PROGRAM Run
VAR	
	buffer					: ARRAY[1..4096] OF BYTE;
	path					: MC_PATH_DATA_REF(ADR(buffer), SIZEOF(buffer));
	
	aTargetPos				: ARRAY[1..cAxesCount] OF MC_LREAL;
	aTransitionParam		: ARRAY[1..2] OF MC_LREAL;
	
	fVelFactor				: LREAL := 1.0;
	
	fbPower					: FB_EnableAxes;
	fbAddAllAxes			: FB_AddAllAxes;
	fbGroupEnable			: MC_GroupEnable;
	fbMoveLinPrep			: MC_MoveLinearAbsolutePreparation;
	fbMovePath				: MC_MovePath;
	fbStop					: MC_GroupStop;
	fbUngroupAxes			: MC_UngroupAllAxes;
	fbGroupReset			: MC_GroupReset;
	fbGroupReadStatus		: MC_GroupReadStatus;
	fbGroupSetOvr			: MC_GroupSetOverride;
	
	nState					: INT := -5;
	nNextState				: INT;
	bMovePrepError			: BOOL;
	bPickCycle				: BOOL;
	bExecutePath			: BOOL := TRUE;
	
	bUserIncrementStep		: BOOL; // user can go to next step
	bUserInfiniteMovement 	: BOOL := TRUE; // user can decide if only one movement is executed or infinite movement.
	bUserStop				: BOOL; // user triggered stop
	bUserForceUngroup		: BOOL; // user triggered ungroup axes
	bUserForceReset			: BOOL; // user triggered reset
	
	
	
	
	bUserEnableAxes:	BOOL:= TRUE;
	bUserConfigGroup:	BOOL	:= FALSE;
	bUserCartesianMode:	BOOL	:= TRUE;
	bUserResetKinGroup:	BOOL	:= FALSE;		
	
	in_stKinToPlc	AT %I*:	NcToPlc_NciChannel_Ref;
	in_stItpToPlc	AT %I*:	NcToPlc_NciChannel_Ref;
	out_stPlcToKin	AT %Q*:	PLCTONC_NCICHANNEL_REF;
	out_stPlcToItp	AT %Q*:	PLCTONC_NCICHANNEL_REF;
	
	//:	FB_EnableAxes;
	bAllAxesReady:	BOOL;
	
	stAxesConfig:	ST_KinAxes;
	fbConfigKinGroup:	FB_KinConfigGroup;
	fbResetKinGroup:	FB_KinResetGroup;
	
	//MODDED CODE VARIABLES
	frameHome : StructFrame := (rXpos := 0, rXpos := 0, rZpos := 147.0, sAlias := 'Home');
	iFrameSequence : INT := 0;
	bRunSequence: BOOL;
	
	
	//////////////
	//Reset
	bResetNC: BOOL;
	bKinFactoryReset: BOOL;
	bResetKinGrp: BOOL;
	nReset: INT;
	nKinReset: INT;
	nGroupReset: INT;
	bKinResetDone: BOOL;
	bGroupResetDone: BOOL;
	fbNCReset	: FB_NCReset;
	bInitMove : BOOL := TRUE;
	iInterpolation : INT := 1;
	bRepeat : BOOL := FALSE;
	
	timerDisable: TON;
	bMagnet: BOOL;
	bXbox : BOOL;
	controller: xbox;
	frameNow: StructFrame;
	frameTarget: StructFrame;
	bAnyBtn : BOOL;
END_VAR

VAR_INPUT
	arrangedFrames : ARRAY [0..20] OF StructFrame;
	nManual: INT;
END_VAR

//==========================================
// PnpSimpleSample V1.3
//==========================================

//==========================================
//	Set variable bUserIncrementStep:= TRUE to go to the next step
//	Variable bUserInfiniteMovement defines if only one movement or infinite
//	movement is executed.
//==========================================



fbGroupReadStatus(
	AxesGroup:= stGroupRef , 
	Enable:= TRUE , 
	Valid=> , 
	Busy=> , 
	GroupMoving=> , 
	GroupHoming=> , 
	GroupErrorStop=> , 
	GroupNotReady=> , 
	GroupStandby=> , 
	GroupStopping=> , 
	GroupDisabled=> , 
	Error=> , 
	ErrorId=> );
IF fbGroupReadStatus.Error THEN
	nState := 9998;
ELSIF NOT fbGroupReadStatus.Valid THEN
	nState := 9999;	
END_IF

fbGroupSetOvr(
	AxesGroup:= stGroupRef, 
	Enable:= TRUE, 
	VelFactor:= fVelFactor , 
	Enabled=> , 
	Busy=> , 
	Error=> , 
	ErrorId=> , 
	ActualVelFactor=> );

IF fbGroupSetOvr.Error THEN
	nState := 9999;
END_IF
	
	


fbPower(
	io_X:= stAxis[1],
	io_Y:= stAxis[2],
	io_Z:= stAxis[3],
	//io_C:= stAxis[4],
	io_M1:= stACSAxis[1],
	io_M2:= stACSAxis[2],
	io_M3:= stACSAxis[3],);
	

stAxesConfig.nAxisIdsAcs[1]	:= stACSAxis[1].NcToPlc.AxisId;
stAxesConfig.nAxisIdsAcs[2]	:= stACSAxis[2].NcToPlc.AxisId;
stAxesConfig.nAxisIdsAcs[3]	:= stACSAxis[3].NcToPlc.AxisId;
stAxesConfig.nAxisIdsMcs[1]	:= stAxis[1].NcToPlc.AxisId;
stAxesConfig.nAxisIdsMcs[2]	:= stAxis[2].NcToPlc.AxisId;
stAxesConfig.nAxisIdsMcs[3]	:= stAxis[3].NcToPlc.AxisId;	
	

CASE nState OF
-5:
	IF bUserIncrementStep THEN
		nNextState := nState +1; 
		nState := 101;
		fbAddAllAxes(Execute:= FALSE);
		fbGroupEnable(AxesGroup:=stGroupRef , Execute:=FALSE);
		fbMovePath(AxesGroup:=stGroupRef ,PathData:=path ,Execute:= FALSE);
		bMovePrepError := FALSE;
	END_IF
-4:	
	fbPower.bEnableAxes := TRUE;
	
	IF fbPower.bAllAxesReady THEN
		IF bUserIncrementStep THEN
			nNextState := nState +1;
			nState := 101;
		END_IF
	ELSIF	fbPower.Error THEN
		nState := nState +1000;	
	END_IF
	
-3:
	fbConfigKinGroup(
		bExecute:=bUserConfigGroup , 
		bCartesianMode:=bUserCartesianMode , 
		stAxesList:=stAxesConfig , 
		stKinRefIn:= in_stKinToPlc, 
		bBusy=> , 
		bDone=> , 
		bError=> , 
		nErrorId=> );
	
	fbResetKinGroup(
		bExecute:=bUserResetKinGroup, 
		nItpChannelId:=0 , 
		stKinRefIn:=in_stKinToPlc, 
		stAxesList:=stAxesConfig, 
		bBusy=> , 
		bDone=> , 
		bError=> , 
		nErrorId=> );
		
	IF fbConfigKinGroup.bDone AND fbResetKinGroup.bDone THEN
		nNextState:= nState + 1;
		nState:= 101;
	ELSIF fbConfigKinGroup.bError OR fbResetKinGroup.bError THEN
		nState:= nState + 1000;
	END_IF
	
-2:
	//Add all axes to group
	fbAddAllAxes(Execute:= TRUE);
	
	IF fbAddAllAxes.Done THEN
		IF bUserIncrementStep THEN
			fbAddAllAxes(Execute:= FALSE);
			nNextState := nState +1;
			nState := 101;
		END_IF
	ELSIF fbAddAllAxes.Error THEN
		nState := nState +1000;
	END_IF
	
-1:	
	//Enable Group
	fbGroupEnable(AxesGroup:=stGroupRef , Execute:=TRUE);
	 
	IF fbGroupEnable.Done THEN
		IF bUserIncrementStep THEN
			fbGroupEnable(AxesGroup:=stGroupRef , Execute:=FALSE);
			nNextState := nState +1;
			nState := 101;
		END_IF
	ELSIF fbGroupEnable.Error THEN
		nState := nState +1000;
	END_IF
0:
	//Fill path table and start execution with fbMovePath
	IF bUserIncrementStep OR bUserInfiniteMovement THEN
		(*IF bPickCycle THEN 
			//Prepare table (MC_MoveLinearAbsolutePreparation)
			A_PreparePathPick();
		ELSE
			//Prepare table (MC_MoveLinearAbsolutePreparation)	
			A_PreparePathPlace();
		END_IF		
		bPickCycle := NOT bPickCycle;*)
		IF bRunSequence THEN
			frameNow.rXpos  := GVL.stAxis[1].NcToPlc.ActPos;
			frameNow.rYpos  := GVL.stAxis[2].NcToPlc.ActPos;
			frameNow.rZpos  := GVL.stAxis[3].NcToPlc.ActPos;
			frameTarget := frameNow;
			END_IF
			
			IF controller.bDpadUp THEN
				//frameTarget := frameNow;
				frameTarget.rYpos := frameNow.rYpos + 1;
				END_IF
			
			IF controller.bDpadDown THEN
				//frameTarget := frameNow;
				frameTarget.rYpos := frameNow.rYpos - 1;
				END_IF
			
			IF controller.bDpadLeft THEN
				//frameTarget := frameNow;
				frameTarget.rXpos := frameNow.rXpos + 1;
				END_IF
			
			IF controller.bDpadRight THEN
				//frameTarget := frameNow;
				frameTarget.rXpos := frameNow.rXpos - 1;
				END_IF
				
			IF controller.bYbtn THEN
				//frameTarget := frameNow;
				frameTarget.rZpos := frameNow.rZpos + 1;
				END_IF
				
			IF controller.bAbtn THEN
				//frameTarget := frameNow;
				frameTarget.rZpos := frameNow.rZpos - 1;
				END_IF
				
			bAnyBtn := (controller.bDpadDown OR controller.bDpadLeft OR controller.bDpadUp OR
						 controller.bDpadRight OR controller.bYbtn OR controller.bAbtn);
			
			IF bAnyBtn THEN
				MoveToPositionGeneral(currentFrame := frameNow, targetFrame := frameTarget, interpolation := 1);
				fbMovePath(AxesGroup:= stGroupRef, PathData:= path, Execute:= TRUE);

				IF bMovePrepError THEN
					nState := nState +1000;
				ELSE
					IF fbMovePath.Done THEN
						fbMovePath(AxesGroup:= stGroupRef, PathData:= path, Execute:= FALSE);
						IF bUserInfiniteMovement THEN
							nState := nState +1;
						ELSIF bUserIncrementStep THEN
							nNextState := nState + 1;
							nState := 101;
						END_IF
					END_IF
				END_IF	
			END_IF			
		END_IF

1:
	//Execute prepared movement
	fbMovePath(
		AxesGroup:= stGroupRef , 
		PathData:= path , 
		Execute:= bExecutePath
	);
	
	IF fbMovePath.Done THEN
		IF bUserIncrementStep THEN
			//ungroup axes
			nNextState := 50;
			nState := 101;
			fbMovePath(AxesGroup:= stGroupRef, PathData:= path, Execute:= FALSE);
		ELSIF bUserInfiniteMovement THEN
			nState := nState -1;
			fbMovePath(AxesGroup:= stGroupRef, PathData:= path, Execute:= FALSE);
		END_IF
	ELSIF fbMovePath.Error THEN
		nState := nState + 1000;	
	END_IF
20:
	fbStop(AxesGroup:=stGroupRef, Execute:= FALSE);
	fbStop(AxesGroup:=stGroupRef, Execute:= TRUE, Jerk:= MC_IGNORE);
	nState := nState + 1;
21:
	fbStop(AxesGroup:=stGroupRef,Execute:= TRUE);
	IF fbStop.Done THEN
		IF bUserIncrementStep THEN
			fbStop(AxesGroup:=stGroupRef, Execute:= FALSE);
			nNextState := 0;
			nState := 101;
		END_IF 		
	ELSIF fbStop.Error THEN
		nState := nState +1000;
	END_IF
50:
	//Disable group and remove all axes 
	fbUngroupAxes(AxesGroup:= stGroupRef, Execute:= FALSE);
	//Check that axes are not moving else we will get a position jump
	IF fbGroupReadStatus.GroupStandby OR fbGroupReadStatus.GroupErrorStop OR fbGroupReadStatus.GroupNotReady THEN
		fbUngroupAxes(AxesGroup:= stGroupRef, Execute:= TRUE);
		nState := nState + 1;
	END_IF	
51:
	fbUngroupAxes(
		AxesGroup:= stGroupRef , 
		Execute:= TRUE, 
		Done=> , 
		Busy=> , 
		Error=> , 
		ErrorId=> );
	
	IF fbUngroupAxes.Done THEN
		IF bUserIncrementStep THEN
			nNextState := -5;
			nState := 101;
		END_IF
	ELSIF fbUngroupAxes.Error THEN
		nState := nState +1000;
	END_IF
80:
	fbGroupReset(AxesGroup:= stGroupRef , Execute:= FALSE);
	fbGroupReset(AxesGroup:= stGroupRef , Execute:= TRUE);
	nState := nState +1;
81:	
	fbGroupReset(
		AxesGroup:= stGroupRef , 
		Execute:= , 
		Done=> , 
		Busy=> , 
		Error=> , 
		ErrorId=> );
	
	IF fbGroupReset.Done THEN
		IF bUserIncrementStep THEN
			IF fbGroupReadStatus.GroupDisabled THEN
				nNextState := -5;
			ELSE
				nNextState := 0;
			END_IF
			nState := 101;
		END_IF				
	END_IF	
101:
	IF (bUserIncrementStep) THEN				
		nState := nNextState;
		bUserIncrementStep := FALSE;
	END_IF
1000..9999:
	;//Error				
END_CASE

IF bUserStop THEN
	nState := 20;
	bUserStop := FALSE;
END_IF
IF bUserForceUngroup THEN
	nState := 50;
	bUserForceUngroup := FALSE;
END_IF
IF bUserForceReset THEN
	nState := 80;
	bUserForceReset := FALSE;
END_IF

ACTION A_AlwaysActive:

fbGroupReadStatus(
	AxesGroup:= stGroupRef , 
	Enable:= TRUE , 
	Valid=> , 
	Busy=> , 
	GroupMoving=> , 
	GroupHoming=> , 
	GroupErrorStop=> , 
	GroupNotReady=> , 
	GroupStandby=> , 
	GroupStopping=> , 
	GroupDisabled=> , 
	Error=> , 
	ErrorId=> );
IF fbGroupReadStatus.Error THEN
	nState := 9998;
ELSIF NOT fbGroupReadStatus.Valid THEN
	nState := 9999;	
END_IF

fbGroupSetOvr(
	AxesGroup:= stGroupRef, 
	Enable:= TRUE, 
	VelFactor:= fVelFactor , 
	Enabled=> , 
	Busy=> , 
	Error=> , 
	ErrorId=> , 
	ActualVelFactor=> );

IF fbGroupSetOvr.Error THEN
	nState := 9999;
END_IF
	
	
fbPower(
	io_X:= stAxis[1],
	io_Y:= stAxis[2],
	io_Z:= stAxis[3],
	io_M1:= stACSAxis[1],
	io_M2:= stACSAxis[2],
	io_M3:= stACSAxis[3]);
	
fbNCReset( 
	bResetDone=> , 
	ResetError=> , 
	io_X:= stAxis[1],     
	io_Y:= stAxis[2],     
	io_Z:= stAxis[3],     
	io_M1:= stACSAxis[1], 
	io_M2:= stACSAxis[2], 
	io_M3:= stACSAxis[3]);	

stAxesConfig.nAxisIdsAcs[1]	:= stACSAxis[1].NcToPlc.AxisId;
stAxesConfig.nAxisIdsAcs[2]	:= stACSAxis[2].NcToPlc.AxisId;
stAxesConfig.nAxisIdsAcs[3]	:= stACSAxis[3].NcToPlc.AxisId;
stAxesConfig.nAxisIdsMcs[1]	:= stAxis[1].NcToPlc.AxisId;
stAxesConfig.nAxisIdsMcs[2]	:= stAxis[2].NcToPlc.AxisId;
stAxesConfig.nAxisIdsMcs[3]	:= stAxis[3].NcToPlc.AxisId;	
	
timerDisable();
END_ACTION

ACTION A_EnableManualMovement:

	fbPower.bEnableAxes := FALSE;
	timerDisable(IN:= TRUE, PT:= T#20MS, Q=> , ET=> );
	IF timerDisable.Q THEN
		fbPower.fOverride := 0;
		fbPower.bEnableAxes := TRUE;
		timerDisable(IN:=FALSE);
		fbNCReset.bReset:=TRUE;
		MAIN.bPowerDisable := FALSE;
	END_IF
END_ACTION

ACTION A_HomePosition:
path.ClearPath();  //Clear nodes that were in path

fbMoveLinPrep.Position						:= ADR(aTargetPos); //pointer to position array
fbMoveLinPrep.PositionCount 				:= cAxesCount; //number of axes in group
fbMoveLinPrep.TransitionParameter			:= ADR (aTransitionParam); //pointer to transition parameter array
fbMoveLinPrep.TransitionParameterCount		:= 2; //number of transition parameters, has to be set always 2
fbMoveLinPrep.BufferMode					:= mcBlendingPrevious;
fbMoveLinPrep.TransitionMode				:= mcTransModeCornerDistanceAdvanced;
//Set dynamics to default values of the axes
fbMoveLinPrep.Acceleration					:= MC_DEFAULT;
fbMoveLinPrep.Deceleration					:= MC_DEFAULT;
fbMoveLinPrep.Jerk							:= MC_DEFAULT;

(* I want to interpolate frames by taking current frame and  next frame,
	and split into N sections, how do i retrieve the current frame? *)

//1st node
aTargetPos[1]				:= 0.0;
aTargetPos[2]				:= 0.0;
aTargetPos[3]				:= 147.0;
////aTargetPos[4]			:= 0;
aTransitionParam[1]			:= 0; //blending distance on previous segment, no influence here
aTransitionParam[2]			:= 0; //blending distance on this segment, no influence here
fbMoveLinPrep(PathData:= path , Velocity:= 200, Acceleration:= 30000, Deceleration:= 30000, Jerk:= 100000, InvokeId:= 10);
bMovePrepError := bMovePrepError OR fbMoveLinPrep.Error;

(*
aTargetPos[1]				:= 100;
aTargetPos[2]				:= 100;
aTargetPos[3]				:= -600;
//aTargetPos[4]			:= 90;
aTransitionParam[1]			:= 30; //blending distance on previous segment (InvokeId=10), defines when to leave line
aTransitionParam[2]			:= 45; //blending distance on this segment, defines latest positionn to be back  on line of InovkeId=20 
fbMoveLinPrep(PathData:= path , Velocity:=200, Acceleration:= 30000, Deceleration:= 30000, Jerk:= 100000, InvokeId:= 20); 
bMovePrepError := bMovePrepError OR fbMoveLinPrep.Error;

aTargetPos[1]				:= 100;
aTargetPos[2]				:= 100;
aTargetPos[3]				:= -750;
//aTargetPos[4]			:= 90;
aTransitionParam[1]			:= 30; 
aTransitionParam[2]			:= 35;
fbMoveLinPrep(PathData:= path , Velocity:= 200, Acceleration:= 30000, Deceleration:= 30000, Jerk:= 100000, InvokeId:= 30);
bMovePrepError := bMovePrepError OR fbMoveLinPrep.Error; *)
END_ACTION

ACTION A_Init:
fbConfigKinGroup(
			bExecute:=FALSE , 
			bCartesianMode:=FALSE , 
			stAxesList:=stAxesConfig , 
			stKinRefIn:= in_stKinToPlc, 
			bBusy=> , 
			bDone=> , 
			bError=> , 
			nErrorId=> );
			
fbResetKinGroup(
			bExecute:=FALSE, 
			nItpChannelId:= , 
			stKinRefIn:=in_stKinToPlc, 
			stAxesList:=stAxesConfig, 
			bBusy=> , 
			bDone=> , 
			bError=> , 
			nErrorId=> );
			
fbNCReset.bReset := FALSE;			
			
bKinResetDone := FALSE;
bGroupResetDone := FALSE;

//bPlace1_Set1 := bPlace2_Set1 := bPlace3_Set1 := bPlace4_Set1:= bPlace5_Set1:= bPlace1_Set2 := bPlace2_Set2 := bPlace3_Set2 := bPlace4_Set2 := FALSE;

//bMagnet_Place1_Set1 := bMagnet_Place2_Set1 := bMagnet_Place3_Set1 := bMagnet_Place1_Set2 := bMagnet_Place2_Set2 := bMagnet_Place3_Set2 := FALSE;
END_ACTION

ACTION A_PreparePathPick:
path.ClearPath();  //Clear nodes that were in path

fbMoveLinPrep.Position						:= ADR(aTargetPos); //pointer to position array
fbMoveLinPrep.PositionCount 				:= cAxesCount; //number of axes in group
fbMoveLinPrep.TransitionParameter			:= ADR (aTransitionParam); //pointer to transition parameter array
fbMoveLinPrep.TransitionParameterCount		:= 2; //number of transition parameters, has to be set always 2
fbMoveLinPrep.BufferMode					:= mcBlendingPrevious;
fbMoveLinPrep.TransitionMode				:= mcTransModeCornerDistanceAdvanced;
//Set dynamics to default values of the axes
fbMoveLinPrep.Acceleration					:= MC_DEFAULT;
fbMoveLinPrep.Deceleration					:= MC_DEFAULT;
fbMoveLinPrep.Jerk							:= MC_DEFAULT;

//1st node
aTargetPos[1]				:= -100;
aTargetPos[2]				:= -100;
aTargetPos[3]				:= -600;
////aTargetPos[4]			:= 0;
aTransitionParam[1]			:= 0; //blending distance on previous segment, no influence here
aTransitionParam[2]			:= 0; //blending distance on this segment, no influence here
fbMoveLinPrep(PathData:= path , Velocity:= 200, Acceleration:= 30000, Deceleration:= 30000, Jerk:= 100000, InvokeId:= 10);
bMovePrepError := bMovePrepError OR fbMoveLinPrep.Error;

aTargetPos[1]				:= 100;
aTargetPos[2]				:= 100;
aTargetPos[3]				:= -600;
////aTargetPos[4]			:= 90;
aTransitionParam[1]			:= 30; //blending distance on previous segment (InvokeId=10), defines when to leave line
aTransitionParam[2]			:= 45; //blending distance on this segment, defines latest positionn to be back  on line of InovkeId=20 
fbMoveLinPrep(PathData:= path , Velocity:=200, Acceleration:= 30000, Deceleration:= 30000, Jerk:= 100000, InvokeId:= 20); 
bMovePrepError := bMovePrepError OR fbMoveLinPrep.Error;

aTargetPos[1]				:= 100;
aTargetPos[2]				:= 100;
aTargetPos[3]				:= -750;
////aTargetPos[4]			:= 90;
aTransitionParam[1]			:= 30; 
aTransitionParam[2]			:= 35;
fbMoveLinPrep(PathData:= path , Velocity:= 200, Acceleration:= 30000, Deceleration:= 30000, Jerk:= 100000, InvokeId:= 30);
bMovePrepError := bMovePrepError OR fbMoveLinPrep.Error;
END_ACTION

ACTION A_PreparePathPlace:
path.ClearPath(); //Clear nodes that were in path

fbMoveLinPrep.Position						:= ADR(aTargetPos); //pointer to position array
fbMoveLinPrep.PositionCount 				:= cAxesCount; //number of axes in group
fbMoveLinPrep.TransitionParameter			:= ADR (aTransitionParam); //pointer to transition parameter array
fbMoveLinPrep.TransitionParameterCount		:= 2; //number of transition parameters, has to be set always 2
fbMoveLinPrep.BufferMode					:= mcBlendingPrevious;
fbMoveLinPrep.TransitionMode				:= mcTransModeCornerDistanceAdvanced;
fbMoveLinPrep.Acceleration					:= MC_DEFAULT;
fbMoveLinPrep.Deceleration					:= MC_DEFAULT;
fbMoveLinPrep.Jerk							:= MC_DEFAULT;

aTargetPos[1]				:= 100;
aTargetPos[2]				:= 100;
aTargetPos[3]				:= -600;
//aTargetPos[4]			:= 90;
aTransitionParam[1]			:= 0; //blending distance on previous segment, no influence here
aTransitionParam[2]			:= 0; //blending distance on this segment, no influence here
fbMoveLinPrep(PathData:= path , Velocity:= 200, Acceleration:= 30000, Deceleration:= 30000, Jerk:= 100000, InvokeId:= 15);
bMovePrepError := bMovePrepError OR fbMoveLinPrep.Error; 

aTargetPos[1]				:= -100;
aTargetPos[2]				:= -100;
aTargetPos[3]				:= -600;
//aTargetPos[4]			:= 0;
aTransitionParam[1]			:= 30; //blending distance on previous segment (InvokeId=10), defines when to leave line
aTransitionParam[2]			:= 45; //blending distance on this segment, defines latest positionn to be back  on line of InovkeId=20
fbMoveLinPrep(PathData:= path , Velocity:= 200, Acceleration:= 30000, Deceleration:= 30000, Jerk:= 100000, InvokeId:= 25);
bMovePrepError := bMovePrepError OR fbMoveLinPrep.Error;

aTargetPos[1]				:= -100;
aTargetPos[2]				:= -100;
aTargetPos[3]				:= -750;
//aTargetPos[4]			:= 0;
aTransitionParam[1]			:= 30; 
aTransitionParam[2]			:= 35;
fbMoveLinPrep(PathData:= path , Velocity:= 200, Acceleration:= 30000, Deceleration:= 30000, Jerk:= 100000, InvokeId:= 35);
bMovePrepError := bMovePrepError OR fbMoveLinPrep.Error;
END_ACTION

ACTION A_ReadXYZValue:
CASE nManual OF
	
	0:
	A_Init();
	nManual := 10;
	bPickCycle := TRUE;
	fbAddAllAxes(Execute:= FALSE);
	fbGroupEnable(AxesGroup:=stGroupRef , Execute:=FALSE);
	fbMovePath(AxesGroup:=stGroupRef ,PathData:=path ,Execute:= FALSE);
	bMovePrepError := FALSE;

10:	
	fbPower.fOverride := 100.0;
	fbPower.bEnableAxes := TRUE;
	
	IF fbPower.bAllAxesReady THEN
		nManual := 20;
	ELSIF	fbPower.Error THEN
		nState := 90;	
	END_IF
	
20:
	bUserConfigGroup:=TRUE;
	bUserCartesianMode:=TRUE;


	fbConfigKinGroup(
		bExecute:=bUserConfigGroup , 
		bCartesianMode:=bUserCartesianMode , 
		stAxesList:=stAxesConfig , 
		stKinRefIn:= in_stKinToPlc, 
		bBusy=> , 
		bDone=> , 
		bError=> , 
		nErrorId=> );
	

	IF fbConfigKinGroup.bDone THEN
		nManual := 100;
	ELSIF fbConfigKinGroup.bError THEN
		nState:= 90;
	END_IF
	(*
30:
	//Add all axes to group
	fbAddAllAxes(Execute:= TRUE);
	
	IF fbAddAllAxes.Done THEN
		fbAddAllAxes(Execute:= FALSE);
		nManual := 40;
	ELSIF fbAddAllAxes.Error THEN
		nState := 90;
	END_IF
	
40:	
	//Enable Group
	fbGroupEnable(AxesGroup:=stGroupRef , Execute:=TRUE);
	 
	IF fbGroupEnable.Done THEN
			fbGroupEnable(AxesGroup:=stGroupRef , Execute:=FALSE);
			nManual := 50;
	ELSIF fbGroupEnable.Error THEN
		nState := 90;
	END_IF
	*)
END_CASE
END_ACTION

METHOD MoveToPositionGeneral
VAR_INPUT
	currentFrame : StructFrame;
	targetFrame : StructFrame;
	interpolation : INT; // interpolates intermittant frames by n number of times
END_VAR

VAR
	unitVector : StructFrame;
	i: INT;
END_VAR
path.ClearPath();  //Clear nodes that were in path

fbMoveLinPrep.Position						:= ADR(aTargetPos); //pointer to position array
fbMoveLinPrep.PositionCount 				:= cAxesCount; //number of axes in group
fbMoveLinPrep.TransitionParameter			:= ADR (aTransitionParam); //pointer to transition parameter array
fbMoveLinPrep.TransitionParameterCount		:= 2; //number of transition parameters, has to be set always 2
fbMoveLinPrep.BufferMode					:= mcBlendingPrevious;
fbMoveLinPrep.TransitionMode				:= mcTransModeCornerDistanceAdvanced;
//Set dynamics to default values of the axes
fbMoveLinPrep.Acceleration					:= MC_DEFAULT;
fbMoveLinPrep.Deceleration					:= MC_DEFAULT;
fbMoveLinPrep.Jerk							:= MC_DEFAULT;

(* I want to interpolate frames by taking current frame and  next frame,
	and split into N sections, how do i retrieve the current frame? *)
	
unitVector.rXpos := (targetFrame.rXpos - currentFrame.rXpos)/interpolation;
unitVector.rYpos := (targetFrame.rYpos - currentFrame.rYpos)/interpolation;
unitVector.rZpos := (targetFrame.rZpos - currentFrame.rZpos)/interpolation;

FOR i:=0 TO interpolation  DO

	//1st node
	aTargetPos[1]				:= currentFrame.rXpos + i * unitVector.rXpos;
	aTargetPos[2]				:= currentFrame.rYpos + i * unitVector.rYpos;
	aTargetPos[3]				:= currentFrame.rZpos + i * unitVector.rZpos;
	//aTargetPos[4]			:= 0;
	aTransitionParam[1]			:= 0; //blending distance on previous segment, no influence here
	aTransitionParam[2]			:= 0; //blending distance on this segment, no influence here
	fbMoveLinPrep(PathData:= path , Velocity:= GVL.lrSpeed, Acceleration:= GVL.acceleration, Deceleration:= GVL.acceleration, Jerk:= 100000, InvokeId:= 30);
	bMovePrepError := bMovePrepError OR fbMoveLinPrep.Error;
	IF bMovePrepError THEN
		EXIT;
	END_IF

END_FOR


(*
aTargetPos[1]				:= 100;
aTargetPos[2]				:= 100;
aTargetPos[3]				:= -600;
//aTargetPos[4]			:= 90;
aTransitionParam[1]			:= 30; //blending distance on previous segment (InvokeId=10), defines when to leave line
aTransitionParam[2]			:= 45; //blending distance on this segment, defines latest positionn to be back  on line of InovkeId=20 
fbMoveLinPrep(PathData:= path , Velocity:=200, Acceleration:= 30000, Deceleration:= 30000, Jerk:= 100000, InvokeId:= 20); 
bMovePrepError := bMovePrepError OR fbMoveLinPrep.Error;

aTargetPos[1]				:= 100;
aTargetPos[2]				:= 100;
aTargetPos[3]				:= -750;
//aTargetPos[4]			:= 90;
aTransitionParam[1]			:= 30; 
aTransitionParam[2]			:= 35;
fbMoveLinPrep(PathData:= path , Velocity:= 200, Acceleration:= 30000, Deceleration:= 30000, Jerk:= 100000, InvokeId:= 30);
bMovePrepError := bMovePrepError OR fbMoveLinPrep.Error; *)
END_METHOD

METHOD MovetoPositionInit
VAR_INPUT
	targetFrame : StructFrame;
END_VAR
path.ClearPath();  //Clear nodes that were in path

fbMoveLinPrep.Position						:= ADR(aTargetPos); //pointer to position array
fbMoveLinPrep.PositionCount 				:= cAxesCount; //number of axes in group
fbMoveLinPrep.TransitionParameter			:= ADR (aTransitionParam); //pointer to transition parameter array
fbMoveLinPrep.TransitionParameterCount		:= 2; //number of transition parameters, has to be set always 2
fbMoveLinPrep.BufferMode					:= mcBlendingPrevious;
fbMoveLinPrep.TransitionMode				:= mcTransModeCornerDistanceAdvanced;
//Set dynamics to default values of the axes
fbMoveLinPrep.Acceleration					:= MC_DEFAULT;
fbMoveLinPrep.Deceleration					:= MC_DEFAULT;
fbMoveLinPrep.Jerk							:= MC_DEFAULT;

(* I want to interpolate frames by taking current frame and  next frame,
	and split into N sections, how do i retrieve the current frame? *)

//1st node
aTargetPos[1]				:= targetFrame.rXpos;
aTargetPos[2]				:= targetFrame.rYpos;
aTargetPos[3]				:= targetFrame.rZpos;
////aTargetPos[4]			:= 0;
aTransitionParam[1]			:= 0; //blending distance on previous segment, no influence here
aTransitionParam[2]			:= 0; //blending distance on this segment, no influence here
fbMoveLinPrep(PathData:= path , Velocity:= GVL.lrSpeed, Acceleration:= GVL.acceleration, Deceleration:= GVL.acceleration, Jerk:= 100000, InvokeId:= 30);
bMovePrepError := bMovePrepError OR fbMoveLinPrep.Error;
END_METHOD

END_PROGRAM

(* stored: Version 1.1.0.1, ProductVersion 3.1.4024.9
   POU Run: Id {cef6c1f9-2a01-4b71-81db-f7ed4deb6965}, SpecialFunc None
   Action A_AlwaysActive: Id {3c43b632-53f6-4303-bbbe-aa9a180d8791}
   Action A_EnableManualMovement: Id {3d649cdb-6ccc-4b2e-809a-11cfd78aa22c}
   Action A_HomePosition: Id {331ee60d-de71-4795-a0c4-e1e046bc151b}
   Action A_Init: Id {f749017d-fbeb-4a05-85ce-e05ee8ac7e08}
   Action A_PreparePathPick: Id {dcb08973-a115-429b-89e2-ef77d8cbb861}
   Action A_PreparePathPlace: Id {807eb52d-d6c5-48fb-b361-4b935b271568}
   Action A_ReadXYZValue: Id {14ac5f61-ed07-472c-989d-d67bfb40a73c}
   Method MoveToPositionGeneral: Id {e4c5583e-e588-4067-89c4-b1ad8292e8ad}
   Method MovetoPositionInit: Id {e631f7e1-f840-40e1-8bdc-db9837a2d8c3} *)
